// TIA Portal project "Door_Prjct" (V16)

(* hardware
DEVICE "S7300/ET200M station_1"  S7-300 station
   slot 0: "Rail_0"  Rail  6ES7 390-1***0-0AA0
   slot 2: "PLC_1"  CPU 314C-2 PN/DP  6ES7 314-6EH04-0AB0  V3.3
      slot 2: "PROFINET interface_1"  PN-IO
         slot 1: "Port_1"  Port
         slot 2: "Port_2"  Port
      slot 5: "DI 24/DO 16_1"  DI24/DO16
      slot 6: "AI 5/AO 2_1"  AI5/AO2
      slot 7: "Count_1"  Counter
      slot 8: "Positioning_1"  Positioning
*)

// ===== PLC "PLC_1"  CPU 314C-2 PN/DP =====

VAR_GLOBAL   // PLC tag table "Default tag table"
   "Etage1_left" AT %I5.0 : Bool;
   "Etage1_right" AT %I5.1 : Bool;
   "Etage2_left" AT %I5.2 : Bool;
   "Etage2_right" AT %I5.3 : Bool;
   "Etage3_left" AT %I5.4 : Bool;
   "Etage3_right" AT %I5.5 : Bool;
   "Etage4_left" AT %I5.6 : Bool;
   "Etage4_right" AT %I5.7 : Bool;
   "Etage1" AT %Q0.0 : Bool;
   "Etage2" AT %Q0.1 : Bool;
   "Etage3" AT %Q0.2 : Bool;
   "Etage4" AT %Q0.3 : Bool;
   "programe 01" AT %I6.0 : Bool;
   "programe 02" AT %I6.1 : Bool;
   "Memoir_Program1" AT %M0.0 : Bool;
   "Timer 2min Program 01" AT %T1 : Timer;
   "Outup_ program 1" AT %M16.0 : Bool;
   "Mem_Programe 02" AT %M0.1 : Bool;
   "SR mem" AT %M16.3 : Bool;
   "Button Etage01" AT %M16.1 : Bool;
   "Outpout Etage01" AT %M16.2 : Bool;
   "edge floor 1" AT %M16.4 : Bool;
   "button etage 02" AT %M16.5 : Bool;
   "Tag_1" AT %M16.6 : Bool;
   "out etage02" AT %M16.7 : Bool;
   "edge out 02" AT %M17.0 : Bool;
   "button etage03" AT %M17.1 : Bool;
   "outp etage 3" AT %M17.2 : Bool;
   "Tag_2" AT %M17.3 : Bool;
   "button etage 04" AT %M17.4 : Bool;
   "out etage 04" AT %M17.5 : Bool;
   "Tag_3" AT %M17.6 : Bool;
   "edge etage 04" AT %M17.7 : Bool;
END_VAR

FUNCTION "Program01" : Void   // FC1, FBD
{ S7_Optimized_Access := 'FALSE' }
VERSION : 0.1
// Program 01  click and return in same floor
   VAR_TEMP   // added for the SCL form of the ladder/FBD networks
      _w1 : Bool;
      _s5time1 : S5Time;
   END_VAR
BEGIN

REGION Network 1: Programe 01
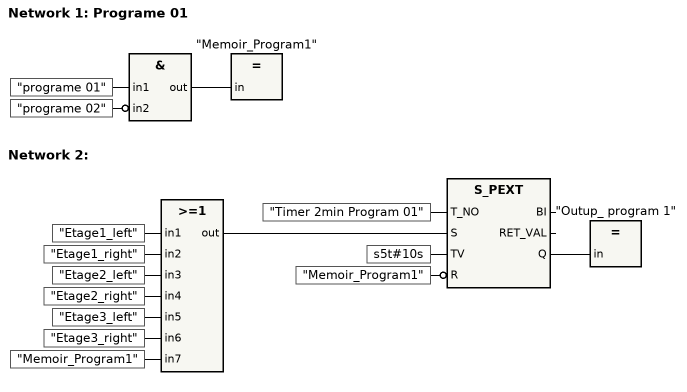
   "Memoir_Program1" := "programe 01" AND NOT "programe 02";
END_REGION

REGION Network 2
   #_s5time1 := S_PEXT(T_NO := "Timer 2min Program 01",
                       S := "Etage1_left" OR "Etage1_right" OR "Etage2_left" OR "Etage2_right" OR "Etage3_left" OR "Etage3_right" OR "Memoir_Program1",
                       TV := s5t#10s,
                       R := NOT "Memoir_Program1",
                       Q => #_w1);
   "Outup_ program 1" := #_w1;
END_REGION
END_FUNCTION

FUNCTION "Program 02" : Void   // FC2, FBD
{ S7_Optimized_Access := 'FALSE' }
VERSION : 0.1
// Programe 02
   VAR_TEMP   // added for the SCL form of the ladder/FBD networks
      _w1 : Bool;
   END_VAR
BEGIN

REGION Network 1: Int Programe 02
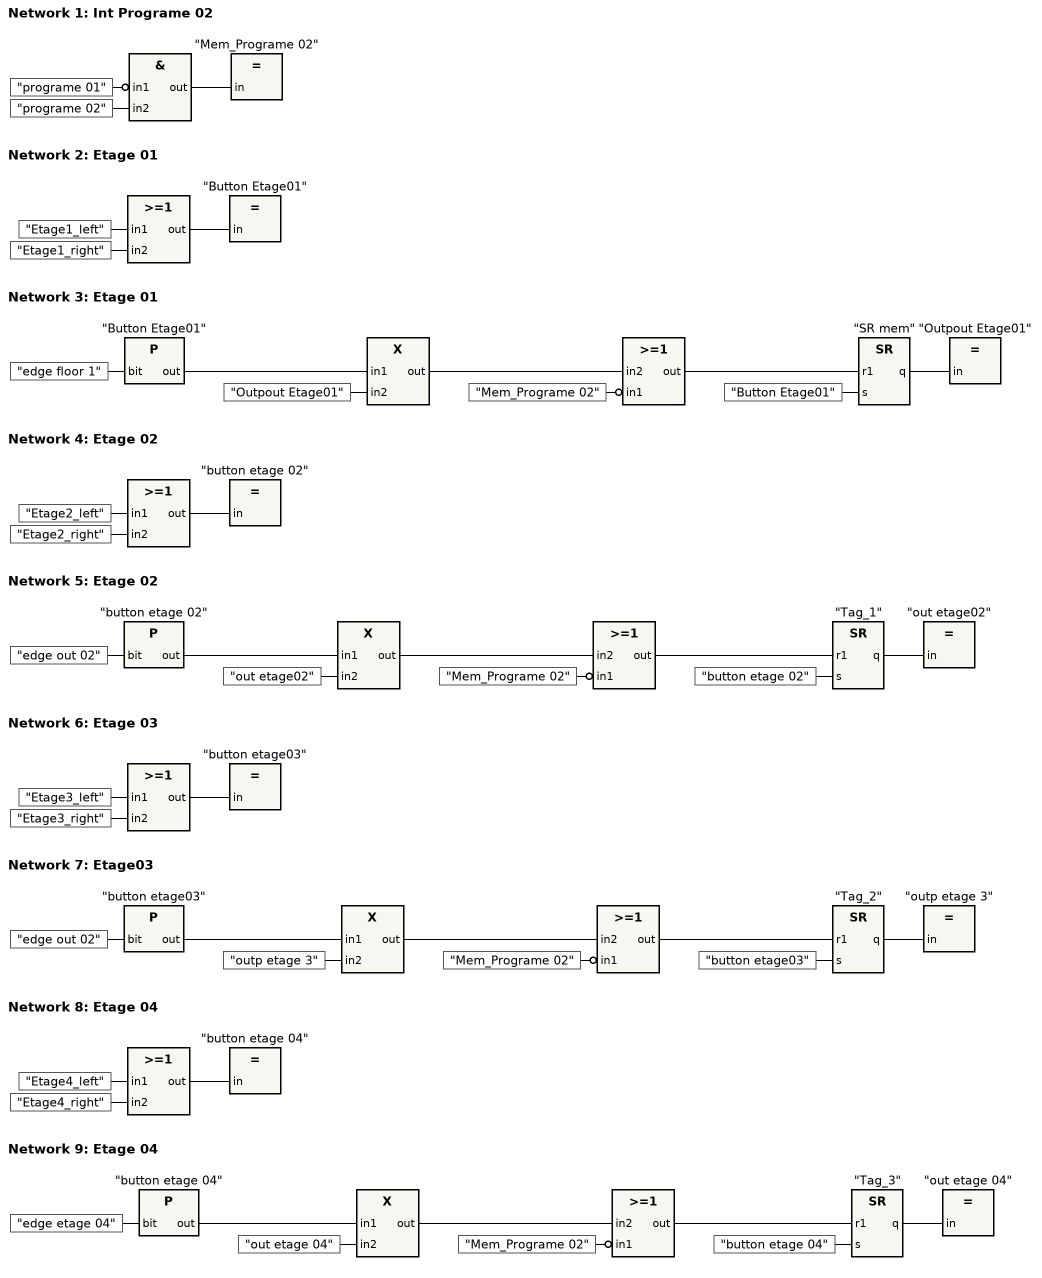
   "Mem_Programe 02" := NOT "programe 01" AND "programe 02";
END_REGION

REGION Network 2: Etage 01
   "Button Etage01" := "Etage1_left" OR "Etage1_right";
END_REGION

REGION Network 3: Etage 01
   #_w1 := "Button Etage01" AND NOT "edge floor 1";   // rising edge of "Button Etage01"
   "edge floor 1" := "Button Etage01";
   IF "Button Etage01" THEN
       "SR mem" := TRUE;   // SR flip-flop
   END_IF;
   IF (#_w1 XOR "Outpout Etage01") OR NOT "Mem_Programe 02" THEN "SR mem" := FALSE; END_IF;
   "Outpout Etage01" := "SR mem";
END_REGION

REGION Network 4: Etage 02
   "button etage 02" := "Etage2_left" OR "Etage2_right";
END_REGION

REGION Network 5: Etage 02
   #_w1 := "button etage 02" AND NOT "edge out 02";   // rising edge of "button etage 02"
   "edge out 02" := "button etage 02";
   IF "button etage 02" THEN
       "Tag_1" := TRUE;   // SR flip-flop
   END_IF;
   IF (#_w1 XOR "out etage02") OR NOT "Mem_Programe 02" THEN "Tag_1" := FALSE; END_IF;
   "out etage02" := "Tag_1";
END_REGION

REGION Network 6: Etage 03
   "button etage03" := "Etage3_left" OR "Etage3_right";
END_REGION

REGION Network 7: Etage03
   #_w1 := "button etage03" AND NOT "edge out 02";   // rising edge of "button etage03"
   "edge out 02" := "button etage03";
   IF "button etage03" THEN
       "Tag_2" := TRUE;   // SR flip-flop
   END_IF;
   IF (#_w1 XOR "outp etage 3") OR NOT "Mem_Programe 02" THEN "Tag_2" := FALSE; END_IF;
   "outp etage 3" := "Tag_2";
END_REGION

REGION Network 8: Etage 04
   "button etage 04" := "Etage4_left" OR "Etage4_right";
END_REGION

REGION Network 9: Etage 04
   #_w1 := "button etage 04" AND NOT "edge etage 04";   // rising edge of "button etage 04"
   "edge etage 04" := "button etage 04";
   IF "button etage 04" THEN
       "Tag_3" := TRUE;   // SR flip-flop
   END_IF;
   IF (#_w1 XOR "out etage 04") OR NOT "Mem_Programe 02" THEN "Tag_3" := FALSE; END_IF;
   "out etage 04" := "Tag_3";
END_REGION
END_FUNCTION

FUNCTION "output" : Void   // FC100, FBD
{ S7_Optimized_Access := 'FALSE' }
VERSION : 0.1
BEGIN

REGION Network 1
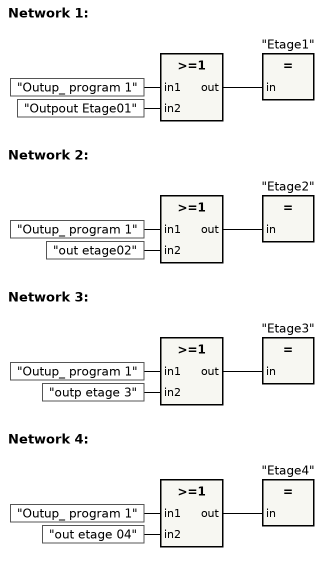
   "Etage1" := "Outup_ program 1" OR "Outpout Etage01";
END_REGION

REGION Network 2
   "Etage2" := "Outup_ program 1" OR "out etage02";
END_REGION

REGION Network 3
   "Etage3" := "Outup_ program 1" OR "outp etage 3";
END_REGION

REGION Network 4
   "Etage4" := "Outup_ program 1" OR "out etage 04";
END_REGION
END_FUNCTION

ORGANIZATION_BLOCK "Main"   // OB1, FBD
TITLE = "Main Program Sweep (Cycle)"
{ S7_Optimized_Access := 'FALSE' }
VERSION : 0.1
   VAR_TEMP
      OB1_EV_CLASS : Byte;   // Bits 0-3 = 1 (Coming event), Bits 4-7 = 1 (Event class 1)
      OB1_SCAN_1 : Byte;   // 1 (Cold restart scan 1 of OB 1), 3 (Scan 2-n of OB 1)
      OB1_PRIORITY : Byte;   // Priority of OB Execution
      OB1_OB_NUMBR : Byte;   // 1 (Organization block 1, OB1)
      OB1_RESERVED_1 : Byte;   // Reserved for system
      OB1_RESERVED_2 : Byte;   // Reserved for system
      OB1_PREV_CYCLE : Int;   // Cycle time of previous OB1 scan (milliseconds)
      OB1_MIN_CYCLE : Int;   // Minimum cycle time of OB1 (milliseconds)
      OB1_MAX_CYCLE : Int;   // Maximum cycle time of OB1 (milliseconds)
      OB1_DATE_TIME : Date_And_Time;   // Date and time OB1 started
   END_VAR
BEGIN

REGION Network 1: P01
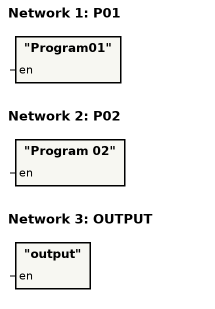
   "Program01"();
END_REGION

REGION Network 2: P02
   "Program 02"();
END_REGION

REGION Network 3: OUTPUT
   "output"();
END_REGION
END_ORGANIZATION_BLOCK